// TIA Portal V19 export
FUNCTION "@MFG TRANSFER LOAD CALCULATE PV" : Void   // FC24, LAD
{ S7_Optimized_Access := 'TRUE' }
// stored: SetENOAutomatically false
   VAR_INPUT
      "MODE SELECTION" : Int;
      "AUTO TRANSFER_1" : Int;
      "AUTO TRANSFER_2" : Int;
      "AUTO TRANSFER_3" : Int;
      "AUTO TRANSFER_4" : Int;
      "AUTO TRANSFER_5" : Int;
      "AUTO TRANSFER_6" : Int;
      "MOVE PV LOAD CELL" : Real;
      "LOAD CELL PV" : Real;
   END_VAR
   VAR_OUTPUT
      MANUAL : Real;
      "MFG TO STORAGE-1 WITH INLINE HOMO" : Real;
      "MFG TO STORAGE-1 WITH INLINE FILTER PRES" : Real;
      "MFG TO STORAGE-2 WITH INLINE HOMO" : Real;
      "MFG TO STORAGE-2 WITH INLINE FILTER PRES" : Real;
      "MFG TO STORAGE-3 WITH INLINE HOMO" : Real;
      "MFG TO STORAGE-3 WITH INLINE FILTER PRES" : Real;
   END_VAR
   VAR_TEMP   // added for the SCL form of the ladder/FBD networks
      _w1 : Bool;
   END_VAR
BEGIN

REGION Network 1: MANUAL
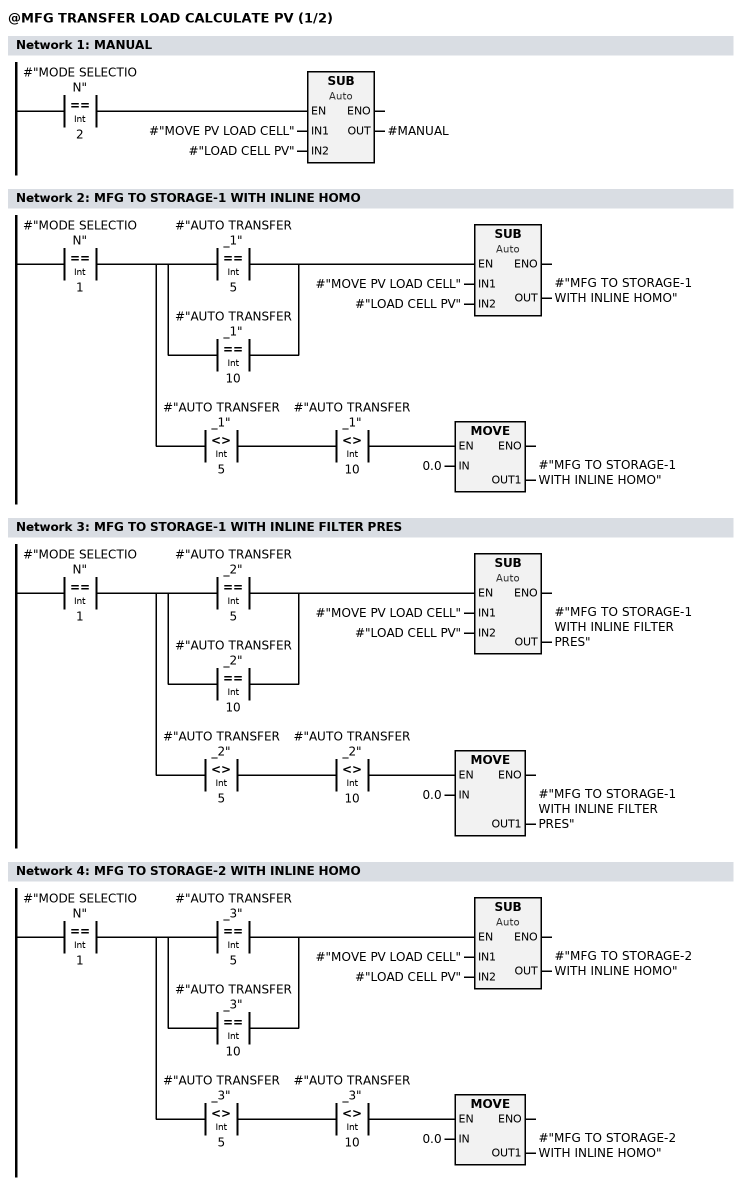
   RUNG wire#powerrail
      { S7_Templates := "SrcType := Int" } EQ_Contact(in1 := #"MODE SELECTION", in2 := 2)
      Sub(in1 := #"MOVE PV LOAD CELL", in2 := #"LOAD CELL PV", out => #MANUAL)
   END_RUNG
   // the same network as SCL:
   IF #"MODE SELECTION" = 2 THEN #MANUAL := #"MOVE PV LOAD CELL" - #"LOAD CELL PV"; END_IF;
END_REGION

REGION Network 2: MFG TO STORAGE-1 WITH INLINE HOMO
   RUNG wire#powerrail
      { S7_Templates := "SrcType := Int" } EQ_Contact(in1 := #"MODE SELECTION", in2 := 1)
      wire#w1
      { S7_Templates := "SrcType := Int" } EQ_Contact(in1 := #"AUTO TRANSFER_1", in2 := 5)
      wire#w2
      Sub(in1 := #"MOVE PV LOAD CELL", in2 := #"LOAD CELL PV", out => #"MFG TO STORAGE-1 WITH INLINE HOMO")
   END_RUNG
   RUNG wire#w1
      { S7_Templates := "SrcType := Int" } EQ_Contact(in1 := #"AUTO TRANSFER_1", in2 := 10)
   END_RUNG wire#w2
   RUNG wire#w1
      { S7_Templates := "SrcType := Int" } NE_Contact(in1 := #"AUTO TRANSFER_1", in2 := 5)
      { S7_Templates := "SrcType := Int" } NE_Contact(in1 := #"AUTO TRANSFER_1", in2 := 10)
      Move(in := 0.0, out1 => #"MFG TO STORAGE-1 WITH INLINE HOMO")
   END_RUNG
   // the same network as SCL:
   #_w1 := #"MODE SELECTION" = 1;
   IF #_w1 AND ((#"AUTO TRANSFER_1" = 5) OR (#"AUTO TRANSFER_1" = 10)) THEN
       #"MFG TO STORAGE-1 WITH INLINE HOMO" := #"MOVE PV LOAD CELL" - #"LOAD CELL PV";
   END_IF;
   IF #_w1 AND (#"AUTO TRANSFER_1" <> 5) AND (#"AUTO TRANSFER_1" <> 10) THEN
       #"MFG TO STORAGE-1 WITH INLINE HOMO" := 0.0;
   END_IF;
END_REGION

REGION Network 3: MFG TO STORAGE-1 WITH INLINE FILTER PRES
   RUNG wire#powerrail
      { S7_Templates := "SrcType := Int" } EQ_Contact(in1 := #"MODE SELECTION", in2 := 1)
      wire#w1
      { S7_Templates := "SrcType := Int" } EQ_Contact(in1 := #"AUTO TRANSFER_2", in2 := 5)
      wire#w2
      Sub(in1 := #"MOVE PV LOAD CELL", in2 := #"LOAD CELL PV", out => #"MFG TO STORAGE-1 WITH INLINE FILTER PRES")
   END_RUNG
   RUNG wire#w1
      { S7_Templates := "SrcType := Int" } EQ_Contact(in1 := #"AUTO TRANSFER_2", in2 := 10)
   END_RUNG wire#w2
   RUNG wire#w1
      { S7_Templates := "SrcType := Int" } NE_Contact(in1 := #"AUTO TRANSFER_2", in2 := 5)
      { S7_Templates := "SrcType := Int" } NE_Contact(in1 := #"AUTO TRANSFER_2", in2 := 10)
      Move(in := 0.0, out1 => #"MFG TO STORAGE-1 WITH INLINE FILTER PRES")
   END_RUNG
   // the same network as SCL:
   #_w1 := #"MODE SELECTION" = 1;
   IF #_w1 AND ((#"AUTO TRANSFER_2" = 5) OR (#"AUTO TRANSFER_2" = 10)) THEN
       #"MFG TO STORAGE-1 WITH INLINE FILTER PRES" := #"MOVE PV LOAD CELL" - #"LOAD CELL PV";
   END_IF;
   IF #_w1 AND (#"AUTO TRANSFER_2" <> 5) AND (#"AUTO TRANSFER_2" <> 10) THEN
       #"MFG TO STORAGE-1 WITH INLINE FILTER PRES" := 0.0;
   END_IF;
END_REGION

REGION Network 4: MFG TO STORAGE-2 WITH INLINE HOMO
   RUNG wire#powerrail
      { S7_Templates := "SrcType := Int" } EQ_Contact(in1 := #"MODE SELECTION", in2 := 1)
      wire#w1
      { S7_Templates := "SrcType := Int" } EQ_Contact(in1 := #"AUTO TRANSFER_3", in2 := 5)
      wire#w2
      Sub(in1 := #"MOVE PV LOAD CELL", in2 := #"LOAD CELL PV", out => #"MFG TO STORAGE-2 WITH INLINE HOMO")
   END_RUNG
   RUNG wire#w1
      { S7_Templates := "SrcType := Int" } EQ_Contact(in1 := #"AUTO TRANSFER_3", in2 := 10)
   END_RUNG wire#w2
   RUNG wire#w1
      { S7_Templates := "SrcType := Int" } NE_Contact(in1 := #"AUTO TRANSFER_3", in2 := 5)
      { S7_Templates := "SrcType := Int" } NE_Contact(in1 := #"AUTO TRANSFER_3", in2 := 10)
      Move(in := 0.0, out1 => #"MFG TO STORAGE-2 WITH INLINE HOMO")
   END_RUNG
   // the same network as SCL:
   #_w1 := #"MODE SELECTION" = 1;
   IF #_w1 AND ((#"AUTO TRANSFER_3" = 5) OR (#"AUTO TRANSFER_3" = 10)) THEN
       #"MFG TO STORAGE-2 WITH INLINE HOMO" := #"MOVE PV LOAD CELL" - #"LOAD CELL PV";
   END_IF;
   IF #_w1 AND (#"AUTO TRANSFER_3" <> 5) AND (#"AUTO TRANSFER_3" <> 10) THEN
       #"MFG TO STORAGE-2 WITH INLINE HOMO" := 0.0;
   END_IF;
END_REGION

REGION Network 5: MFG TO STORAGE-2 WITH INLINE FILTER PRES
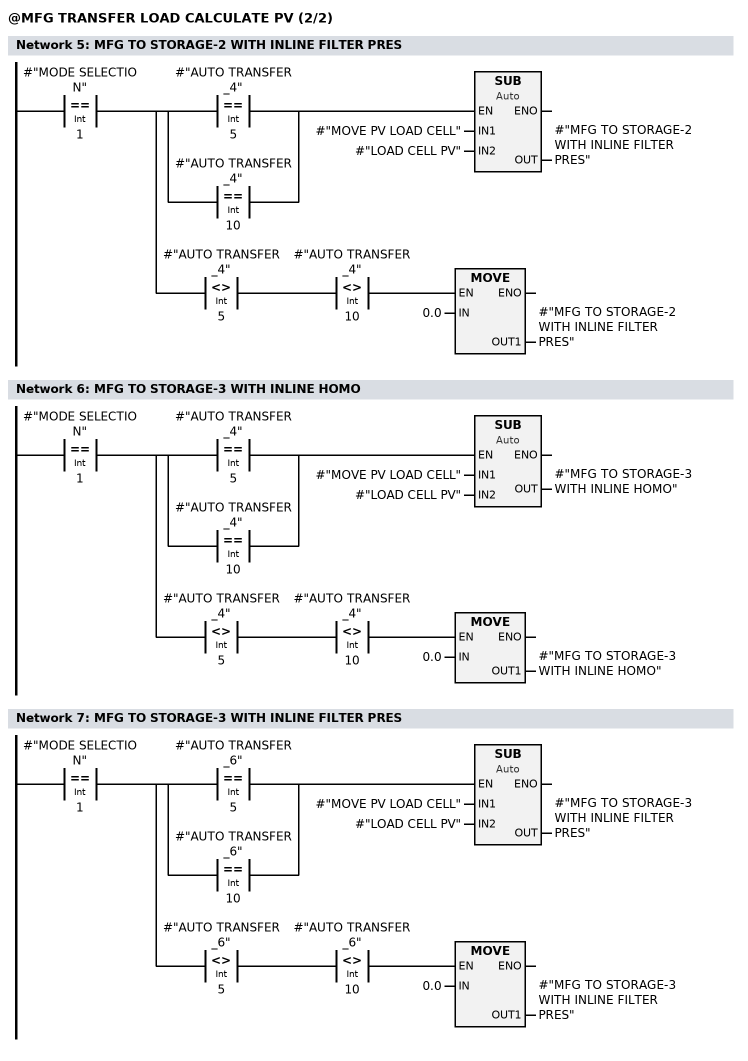
   RUNG wire#powerrail
      { S7_Templates := "SrcType := Int" } EQ_Contact(in1 := #"MODE SELECTION", in2 := 1)
      wire#w1
      { S7_Templates := "SrcType := Int" } EQ_Contact(in1 := #"AUTO TRANSFER_4", in2 := 5)
      wire#w2
      Sub(in1 := #"MOVE PV LOAD CELL", in2 := #"LOAD CELL PV", out => #"MFG TO STORAGE-2 WITH INLINE FILTER PRES")
   END_RUNG
   RUNG wire#w1
      { S7_Templates := "SrcType := Int" } EQ_Contact(in1 := #"AUTO TRANSFER_4", in2 := 10)
   END_RUNG wire#w2
   RUNG wire#w1
      { S7_Templates := "SrcType := Int" } NE_Contact(in1 := #"AUTO TRANSFER_4", in2 := 5)
      { S7_Templates := "SrcType := Int" } NE_Contact(in1 := #"AUTO TRANSFER_4", in2 := 10)
      Move(in := 0.0, out1 => #"MFG TO STORAGE-2 WITH INLINE FILTER PRES")
   END_RUNG
   // the same network as SCL:
   #_w1 := #"MODE SELECTION" = 1;
   IF #_w1 AND ((#"AUTO TRANSFER_4" = 5) OR (#"AUTO TRANSFER_4" = 10)) THEN
       #"MFG TO STORAGE-2 WITH INLINE FILTER PRES" := #"MOVE PV LOAD CELL" - #"LOAD CELL PV";
   END_IF;
   IF #_w1 AND (#"AUTO TRANSFER_4" <> 5) AND (#"AUTO TRANSFER_4" <> 10) THEN
       #"MFG TO STORAGE-2 WITH INLINE FILTER PRES" := 0.0;
   END_IF;
END_REGION

REGION Network 6: MFG TO STORAGE-3 WITH INLINE HOMO
   RUNG wire#powerrail
      { S7_Templates := "SrcType := Int" } EQ_Contact(in1 := #"MODE SELECTION", in2 := 1)
      wire#w1
      { S7_Templates := "SrcType := Int" } EQ_Contact(in1 := #"AUTO TRANSFER_4", in2 := 5)
      wire#w2
      Sub(in1 := #"MOVE PV LOAD CELL", in2 := #"LOAD CELL PV", out => #"MFG TO STORAGE-3 WITH INLINE HOMO")
   END_RUNG
   RUNG wire#w1
      { S7_Templates := "SrcType := Int" } EQ_Contact(in1 := #"AUTO TRANSFER_4", in2 := 10)
   END_RUNG wire#w2
   RUNG wire#w1
      { S7_Templates := "SrcType := Int" } NE_Contact(in1 := #"AUTO TRANSFER_4", in2 := 5)
      { S7_Templates := "SrcType := Int" } NE_Contact(in1 := #"AUTO TRANSFER_4", in2 := 10)
      Move(in := 0.0, out1 => #"MFG TO STORAGE-3 WITH INLINE HOMO")
   END_RUNG
   // the same network as SCL:
   #_w1 := #"MODE SELECTION" = 1;
   IF #_w1 AND ((#"AUTO TRANSFER_4" = 5) OR (#"AUTO TRANSFER_4" = 10)) THEN
       #"MFG TO STORAGE-3 WITH INLINE HOMO" := #"MOVE PV LOAD CELL" - #"LOAD CELL PV";
   END_IF;
   IF #_w1 AND (#"AUTO TRANSFER_4" <> 5) AND (#"AUTO TRANSFER_4" <> 10) THEN
       #"MFG TO STORAGE-3 WITH INLINE HOMO" := 0.0;
   END_IF;
END_REGION

REGION Network 7: MFG TO STORAGE-3 WITH INLINE FILTER PRES
   RUNG wire#powerrail
      { S7_Templates := "SrcType := Int" } EQ_Contact(in1 := #"MODE SELECTION", in2 := 1)
      wire#w1
      { S7_Templates := "SrcType := Int" } EQ_Contact(in1 := #"AUTO TRANSFER_6", in2 := 5)
      wire#w2
      Sub(in1 := #"MOVE PV LOAD CELL", in2 := #"LOAD CELL PV", out => #"MFG TO STORAGE-3 WITH INLINE FILTER PRES")
   END_RUNG
   RUNG wire#w1
      { S7_Templates := "SrcType := Int" } EQ_Contact(in1 := #"AUTO TRANSFER_6", in2 := 10)
   END_RUNG wire#w2
   RUNG wire#w1
      { S7_Templates := "SrcType := Int" } NE_Contact(in1 := #"AUTO TRANSFER_6", in2 := 5)
      { S7_Templates := "SrcType := Int" } NE_Contact(in1 := #"AUTO TRANSFER_6", in2 := 10)
      Move(in := 0.0, out1 => #"MFG TO STORAGE-3 WITH INLINE FILTER PRES")
   END_RUNG
   // the same network as SCL:
   #_w1 := #"MODE SELECTION" = 1;
   IF #_w1 AND ((#"AUTO TRANSFER_6" = 5) OR (#"AUTO TRANSFER_6" = 10)) THEN
       #"MFG TO STORAGE-3 WITH INLINE FILTER PRES" := #"MOVE PV LOAD CELL" - #"LOAD CELL PV";
   END_IF;
   IF #_w1 AND (#"AUTO TRANSFER_6" <> 5) AND (#"AUTO TRANSFER_6" <> 10) THEN
       #"MFG TO STORAGE-3 WITH INLINE FILTER PRES" := 0.0;
   END_IF;
END_REGION
END_FUNCTION
